(* Logix 5000 project; controller R5_CSS vendor 1 type 14 code 74 rev 19.11; software revision 19.01; part 5 of 18 *)
(* tags used below, declared in another part *)
   Coal_Tank_Heel_Inches : REAL;
   Coal_Tank_Height_Inches : REAL;
   ColdBoot : BOOL;
   DisableCommand : BOOL;
   EnableCommand : BOOL;
   Fault : BOOL;
   FirstScanLatch : BOOL;
   FirstScanLatchTON : TIMER;
   HART1 : HARTModuleDef;
   HARTData1 : HARTData;
   HEART_DATA : INT[122];
   IP_Address : DINT[4];
   IP_AddressGetMSG : MESSAGE;
   IP_AddressGetMSG_TON : TIMER;
   IP_AddressSetMSG : MESSAGE;
   LC303A : LEVEL_CONTROL;   // AQUEOUS PHASE OF PRIMARY SETTLER
   LC303A_LT_Raw : REAL;
   LC303B : LEVEL_CONTROL;   // INTERFACE LEVEL OF PRIMARY CONDENSER
   LC303B_LT_Raw : REAL;
   LT303_Probe_Length_Inches : REAL;
   LT303_RAW : REAL[5];   // LT 303 RAW
   LT303_Scale_Param : REAL;
   My_IP_Address : DINT[4];
   My_Subnet : DINT[4];
   P101A : PUMP_CONTROL;
   P101B : PUMP_CONTROL;
   P303A : PUMP_CONTROL;
   P303B : PUMP_CONTROL;
   SetMyIP_Enabled : BOOL;
   TCP_GetAll : TCPGetAllConfig;
   TCP_SetAll : TCPSetAllConfig;
   Test : INT[500];
   WarmBoot : BOOL;
(* MainProgram, continued *)

ROUTINE A2a_MM_HART   (* ladder *)
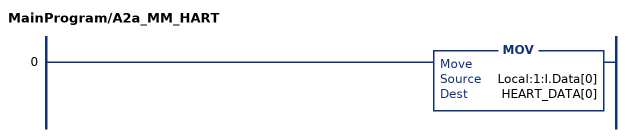
   0: MOV(Local:1:I.Data[0],HEART_DATA[0]);
END_ROUTINE

ROUTINE A2b_HART_READ   (* ladder *)
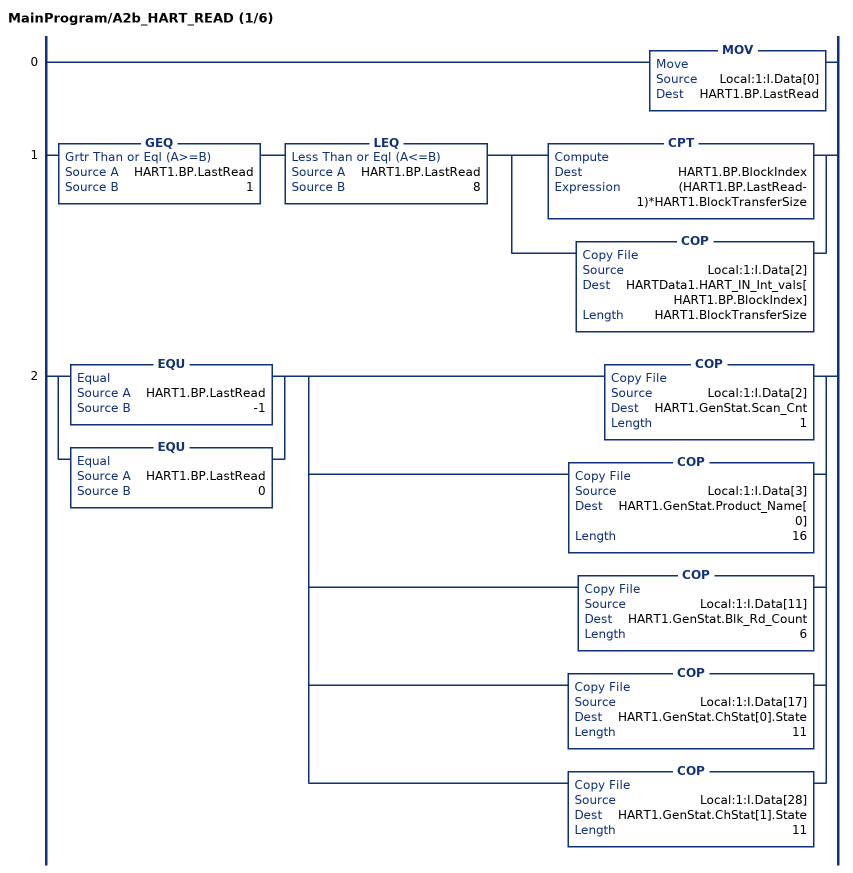
   0: MOV(Local:1:I.Data[0],HART1.BP.LastRead);
   1: GEQ(HART1.BP.LastRead,1)LEQ(HART1.BP.LastRead,8)[CPT(HART1.BP.BlockIndex,(HART1.BP.LastRead-1)*HART1.BlockTransferSize) ,COP(Local:1:I.Data[2],HARTData1.HART_IN_Int_vals[HART1.BP.BlockIndex],HART1.BlockTransferSize) ];
   2: [EQU(HART1.BP.LastRead,-1) ,EQU(HART1.BP.LastRead,0) ][COP(Local:1:I.Data[2],HART1.GenStat.Scan_Cnt,1) ,COP(Local:1:I.Data[3],HART1.GenStat.Product_Name[0],16) ,COP(Local:1:I.Data[11],HART1.GenStat.Blk_Rd_Count,6) ,COP(Local:1:I.Data[17],HART1.GenStat.ChStat[0].State,11) ,COP(Local:1:I.Data[28],HART1.GenStat.ChStat[1].State,11) ];
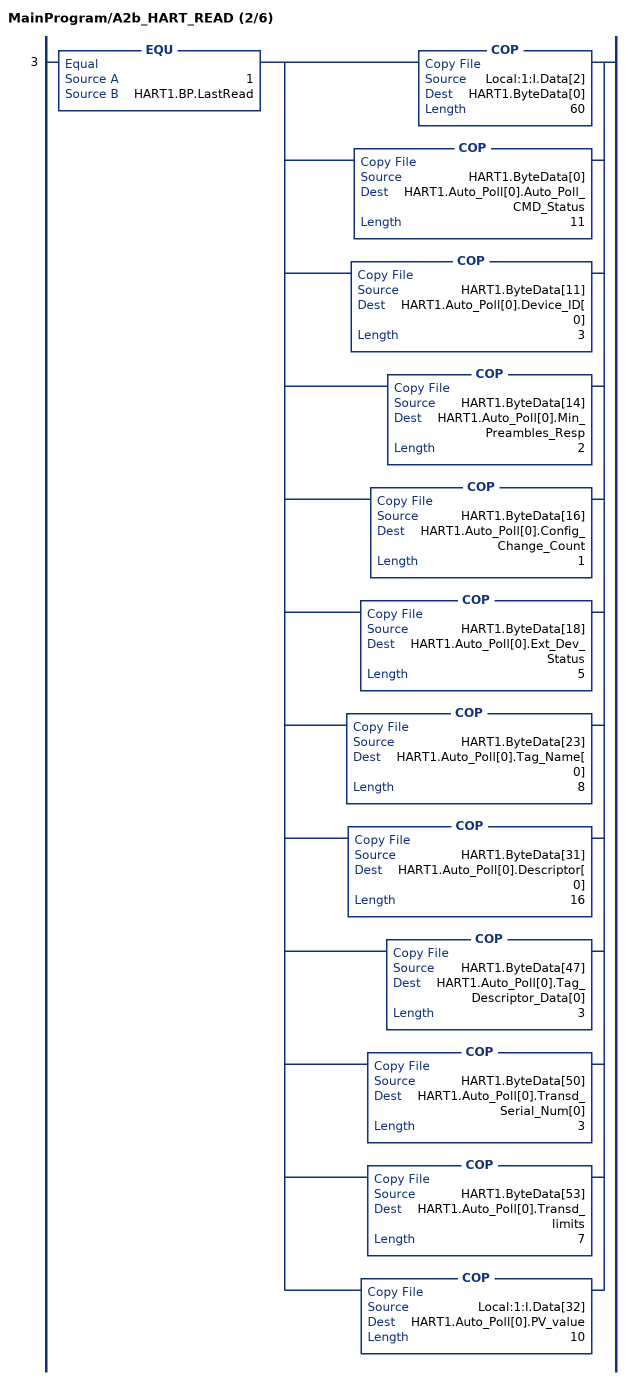
   3: EQU(1,HART1.BP.LastRead)[COP(Local:1:I.Data[2],HART1.ByteData[0],60) ,COP(HART1.ByteData[0],HART1.Auto_Poll[0].Auto_Poll_CMD_Status,11) ,COP(HART1.ByteData[11],HART1.Auto_Poll[0].Device_ID[0],3) ,COP(HART1.ByteData[14],HART1.Auto_Poll[0].Min_Preambles_Resp,2) ,COP(HART1.ByteData[16],HART1.Auto_Poll[0].Config_Change_Count,1) ,COP(HART1.ByteData[18],HART1.Auto_Poll[0].Ext_Dev_Status,5) ,COP(HART1.ByteData[23],HART1.Auto_Poll[0].Tag_Name[0],8) ,COP(HART1.ByteData[31],HART1.Auto_Poll[0].Descriptor[0],16) ,COP(HART1.ByteData[47],HART1.Auto_Poll[0].Tag_Descriptor_Data[0],3) ,COP(HART1.ByteData[50],HART1.Auto_Poll[0].Transd_Serial_Num[0],3) ,COP(HART1.ByteData[53],HART1.Auto_Poll[0].Transd_limits,7) ,COP(Local:1:I.Data[32],HART1.Auto_Poll[0].PV_value,10) ];
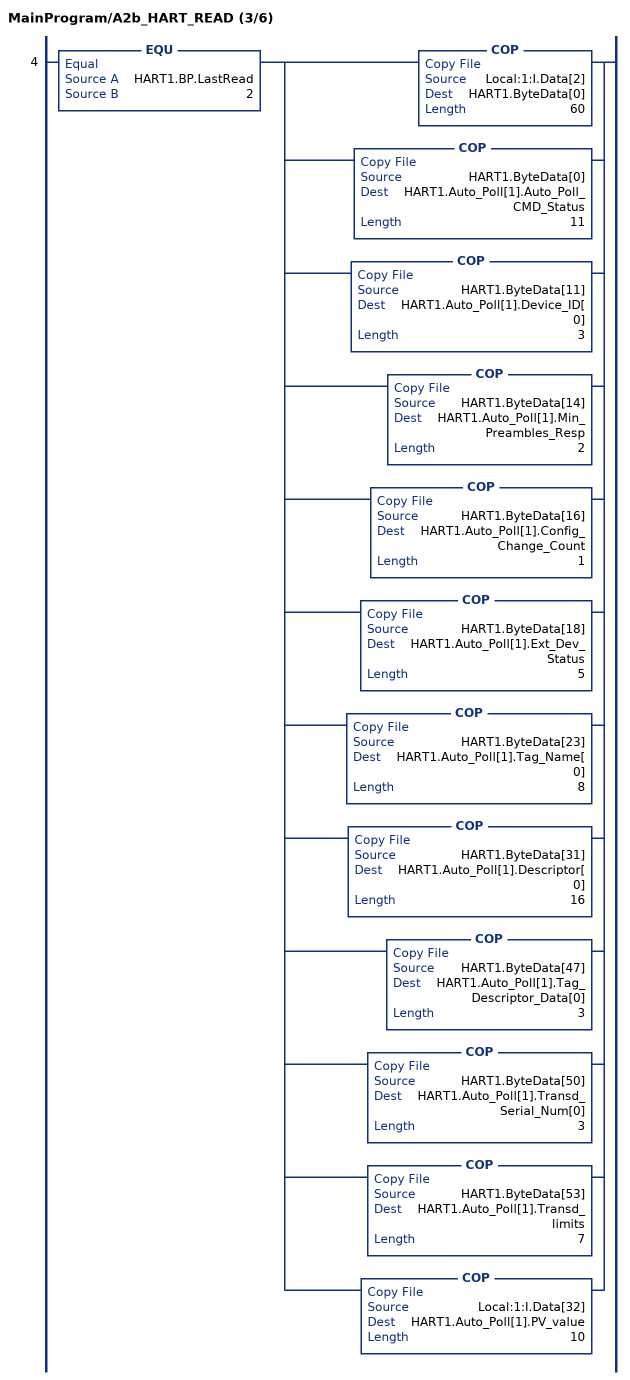
   4: EQU(HART1.BP.LastRead,2)[COP(Local:1:I.Data[2],HART1.ByteData[0],60) ,COP(HART1.ByteData[0],HART1.Auto_Poll[1].Auto_Poll_CMD_Status,11) ,COP(HART1.ByteData[11],HART1.Auto_Poll[1].Device_ID[0],3) ,COP(HART1.ByteData[14],HART1.Auto_Poll[1].Min_Preambles_Resp,2) ,COP(HART1.ByteData[16],HART1.Auto_Poll[1].Config_Change_Count,1) ,COP(HART1.ByteData[18],HART1.Auto_Poll[1].Ext_Dev_Status,5) ,COP(HART1.ByteData[23],HART1.Auto_Poll[1].Tag_Name[0],8) ,COP(HART1.ByteData[31],HART1.Auto_Poll[1].Descriptor[0],16) ,COP(HART1.ByteData[47],HART1.Auto_Poll[1].Tag_Descriptor_Data[0],3) ,COP(HART1.ByteData[50],HART1.Auto_Poll[1].Transd_Serial_Num[0],3) ,COP(HART1.ByteData[53],HART1.Auto_Poll[1].Transd_limits,7) ,COP(Local:1:I.Data[32],HART1.Auto_Poll[1].PV_value,10) ];
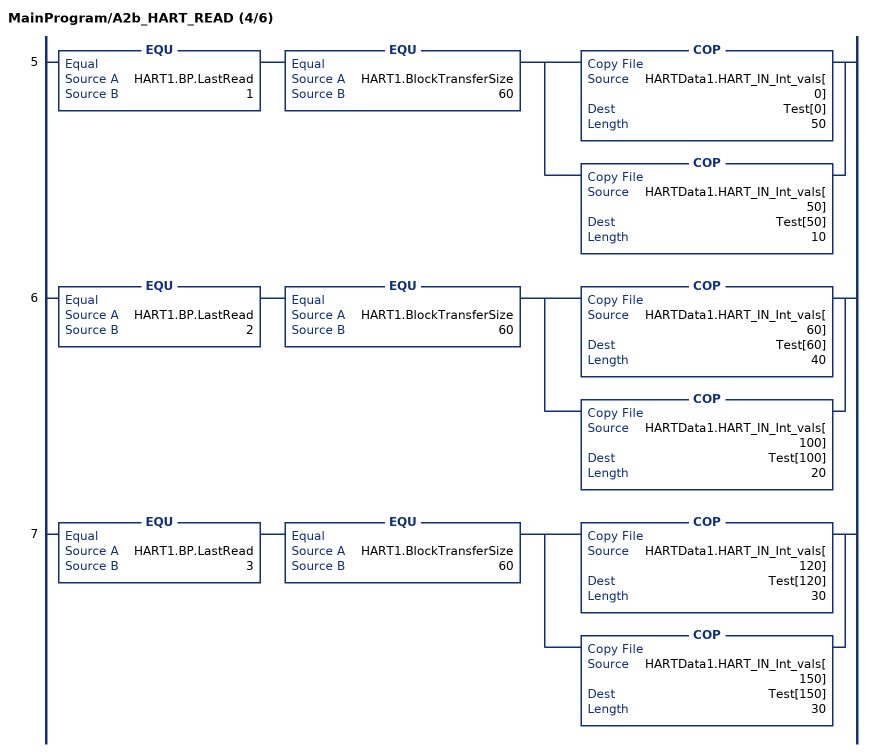
   5: EQU(HART1.BP.LastRead,1)EQU(HART1.BlockTransferSize,60)[COP(HARTData1.HART_IN_Int_vals[0],Test[0],50) ,COP(HARTData1.HART_IN_Int_vals[50],Test[50],10) ];
   6: EQU(HART1.BP.LastRead,2)EQU(HART1.BlockTransferSize,60)[COP(HARTData1.HART_IN_Int_vals[60],Test[60],40) ,COP(HARTData1.HART_IN_Int_vals[100],Test[100],20) ];
   7: EQU(HART1.BP.LastRead,3)EQU(HART1.BlockTransferSize,60)[COP(HARTData1.HART_IN_Int_vals[120],Test[120],30) ,COP(HARTData1.HART_IN_Int_vals[150],Test[150],30) ];
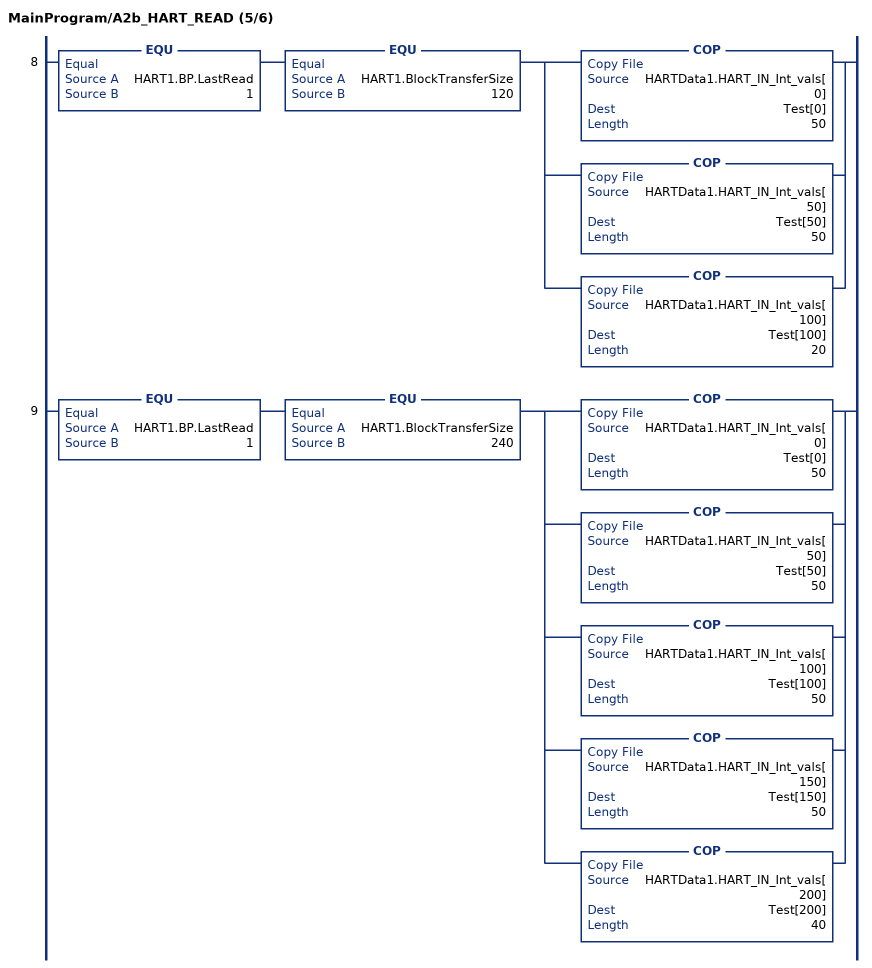
   8: EQU(HART1.BP.LastRead,1)EQU(HART1.BlockTransferSize,120)[COP(HARTData1.HART_IN_Int_vals[0],Test[0],50) ,COP(HARTData1.HART_IN_Int_vals[50],Test[50],50) ,COP(HARTData1.HART_IN_Int_vals[100],Test[100],20) ];
   9: EQU(HART1.BP.LastRead,1)EQU(HART1.BlockTransferSize,240)[COP(HARTData1.HART_IN_Int_vals[0],Test[0],50) ,COP(HARTData1.HART_IN_Int_vals[50],Test[50],50) ,COP(HARTData1.HART_IN_Int_vals[100],Test[100],50) ,COP(HARTData1.HART_IN_Int_vals[150],Test[150],50) ,COP(HARTData1.HART_IN_Int_vals[200],Test[200],40) ];
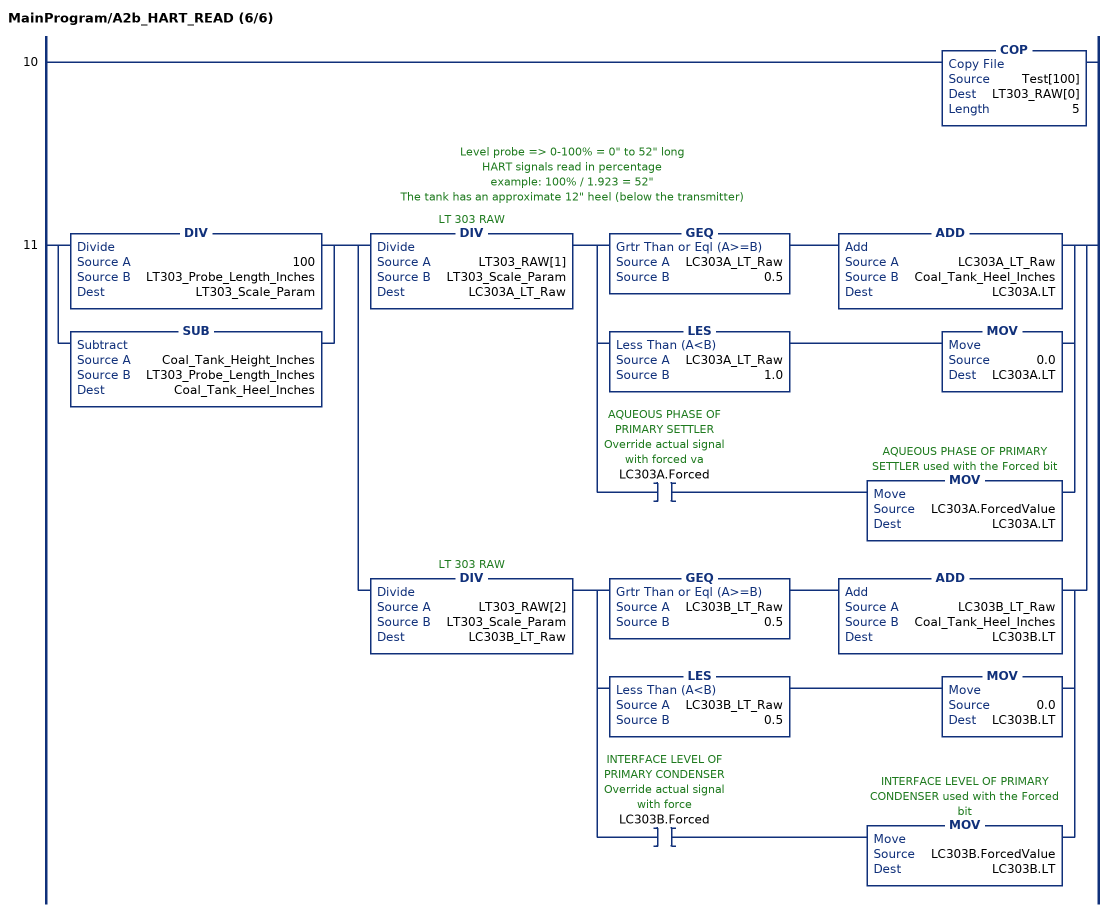
   10: COP(Test[100],LT303_RAW[0],5);
   // Level probe => 0-100% = 0" to 52" long
   // HART signals read in percentage
   // example: 100% / 1.923 = 52"
   // The tank has an approximate 12" heel (below the transmitter)
   11: [DIV(100,LT303_Probe_Length_Inches,LT303_Scale_Param) ,SUB(Coal_Tank_Height_Inches,LT303_Probe_Length_Inches,Coal_Tank_Heel_Inches) ][DIV(LT303_RAW[1],LT303_Scale_Param,LC303A_LT_Raw) [GEQ(LC303A_LT_Raw,0.5) ADD(LC303A_LT_Raw,Coal_Tank_Heel_Inches,LC303A.LT) ,LES(LC303A_LT_Raw,1.0) MOV(0.0,LC303A.LT) ,XIC(LC303A.Forced) MOV(LC303A.ForcedValue,LC303A.LT) ] ,DIV(LT303_RAW[2],LT303_Scale_Param,LC303B_LT_Raw) [GEQ(LC303B_LT_Raw,0.5) ADD(LC303B_LT_Raw,Coal_Tank_Heel_Inches,LC303B.LT) ,LES(LC303B_LT_Raw,0.5) MOV(0.0,LC303B.LT) ,XIC(LC303B.Forced) MOV(LC303B.ForcedValue,LC303B.LT) ] ];
END_ROUTINE

ROUTINE A2c_HART_WRITEE   (* ladder *)
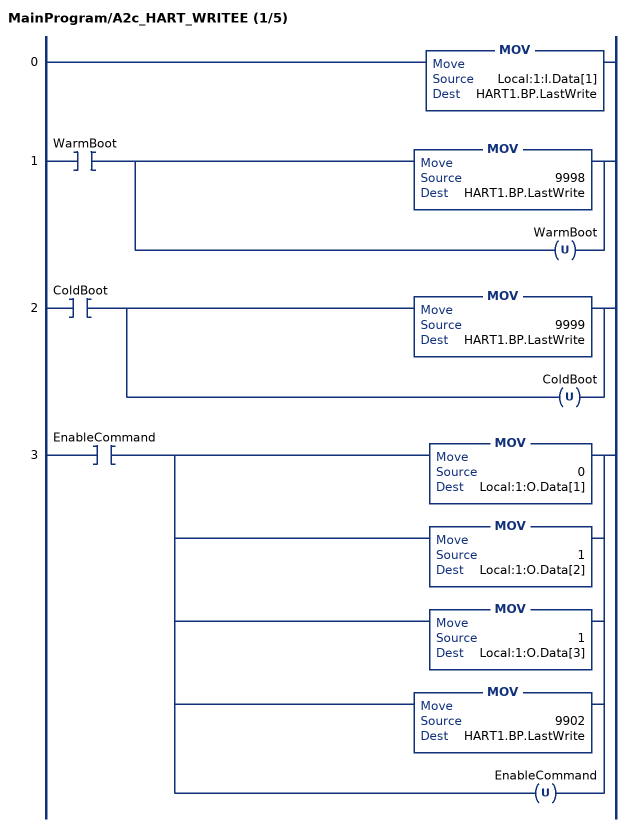
   0: MOV(Local:1:I.Data[1],HART1.BP.LastWrite);
   1: XIC(WarmBoot)[MOV(9998,HART1.BP.LastWrite) ,OTU(WarmBoot) ];
   2: XIC(ColdBoot)[MOV(9999,HART1.BP.LastWrite) ,OTU(ColdBoot) ];
   3: XIC(EnableCommand)[MOV(0,Local:1:O.Data[1]) ,MOV(1,Local:1:O.Data[2]) ,MOV(1,Local:1:O.Data[3]) ,MOV(9902,HART1.BP.LastWrite) ,OTU(EnableCommand) ];
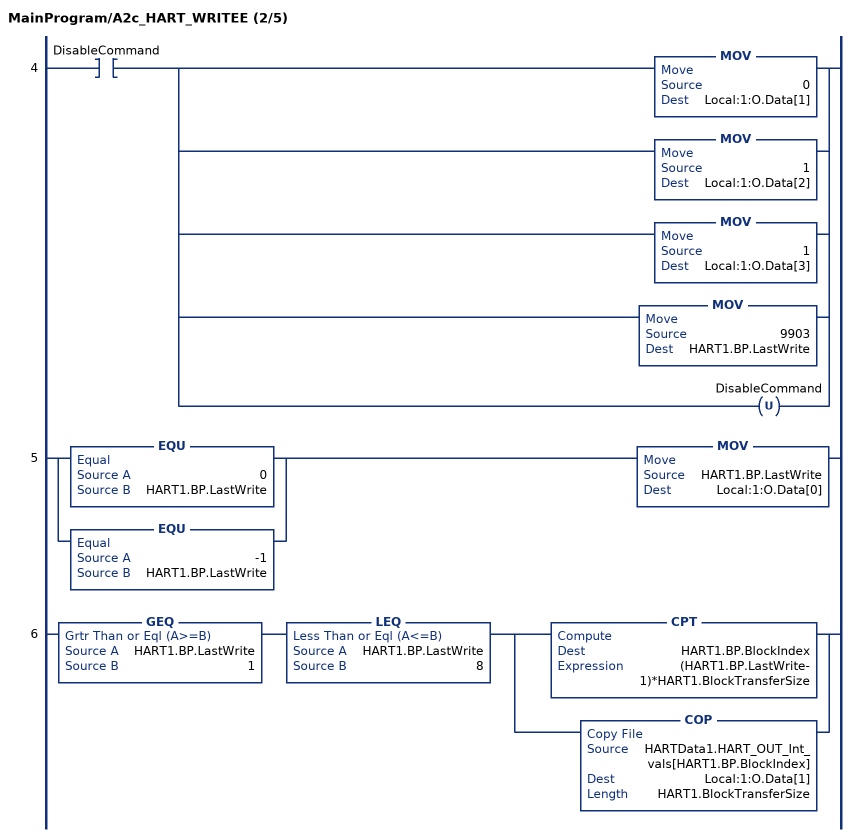
   4: XIC(DisableCommand)[MOV(0,Local:1:O.Data[1]) ,MOV(1,Local:1:O.Data[2]) ,MOV(1,Local:1:O.Data[3]) ,MOV(9903,HART1.BP.LastWrite) ,OTU(DisableCommand) ];
   5: [EQU(0,HART1.BP.LastWrite) ,EQU(-1,HART1.BP.LastWrite) ]MOV(HART1.BP.LastWrite,Local:1:O.Data[0]);
   6: GEQ(HART1.BP.LastWrite,1)LEQ(HART1.BP.LastWrite,8)[CPT(HART1.BP.BlockIndex,(HART1.BP.LastWrite-1)*HART1.BlockTransferSize) ,COP(HARTData1.HART_OUT_Int_vals[HART1.BP.BlockIndex],Local:1:O.Data[1],HART1.BlockTransferSize) ];
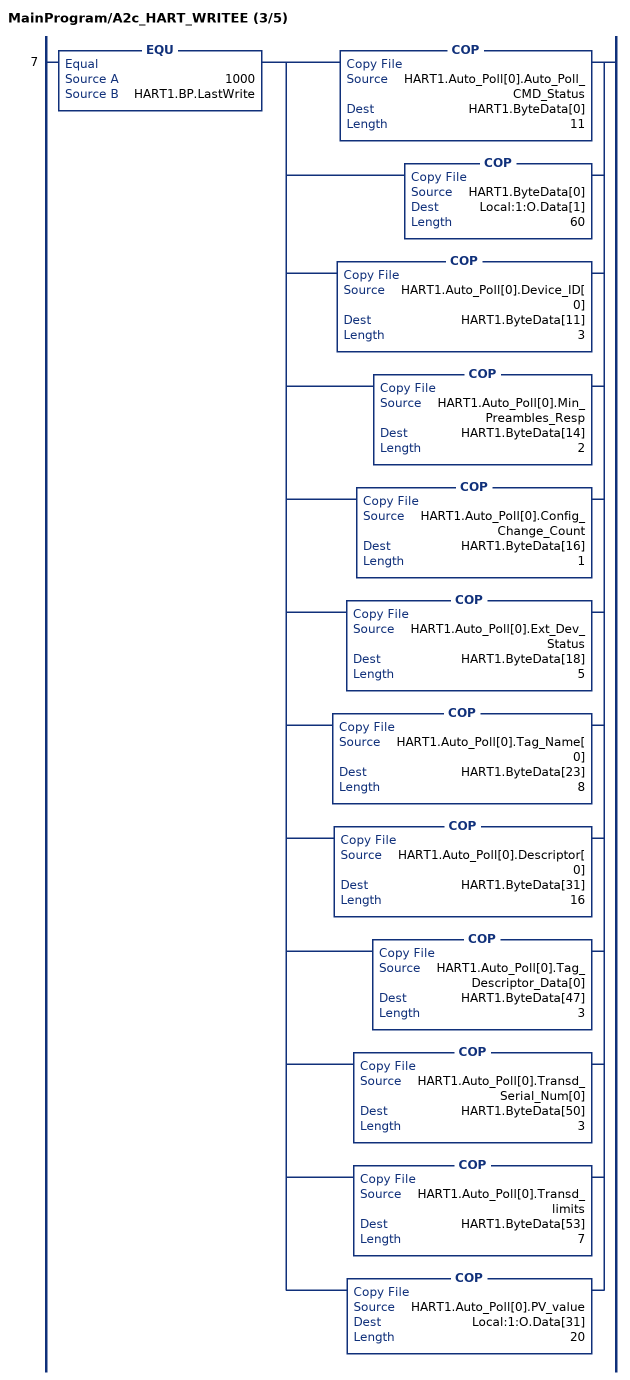
   7: EQU(1000,HART1.BP.LastWrite)[COP(HART1.Auto_Poll[0].Auto_Poll_CMD_Status,HART1.ByteData[0],11) ,COP(HART1.ByteData[0],Local:1:O.Data[1],60) ,COP(HART1.Auto_Poll[0].Device_ID[0],HART1.ByteData[11],3) ,COP(HART1.Auto_Poll[0].Min_Preambles_Resp,HART1.ByteData[14],2) ,COP(HART1.Auto_Poll[0].Config_Change_Count,HART1.ByteData[16],1) ,COP(HART1.Auto_Poll[0].Ext_Dev_Status,HART1.ByteData[18],5) ,COP(HART1.Auto_Poll[0].Tag_Name[0],HART1.ByteData[23],8) ,COP(HART1.Auto_Poll[0].Descriptor[0],HART1.ByteData[31],16) ,COP(HART1.Auto_Poll[0].Tag_Descriptor_Data[0],HART1.ByteData[47],3) ,COP(HART1.Auto_Poll[0].Transd_Serial_Num[0],HART1.ByteData[50],3) ,COP(HART1.Auto_Poll[0].Transd_limits,HART1.ByteData[53],7) ,COP(HART1.Auto_Poll[0].PV_value,Local:1:O.Data[31],20) ];
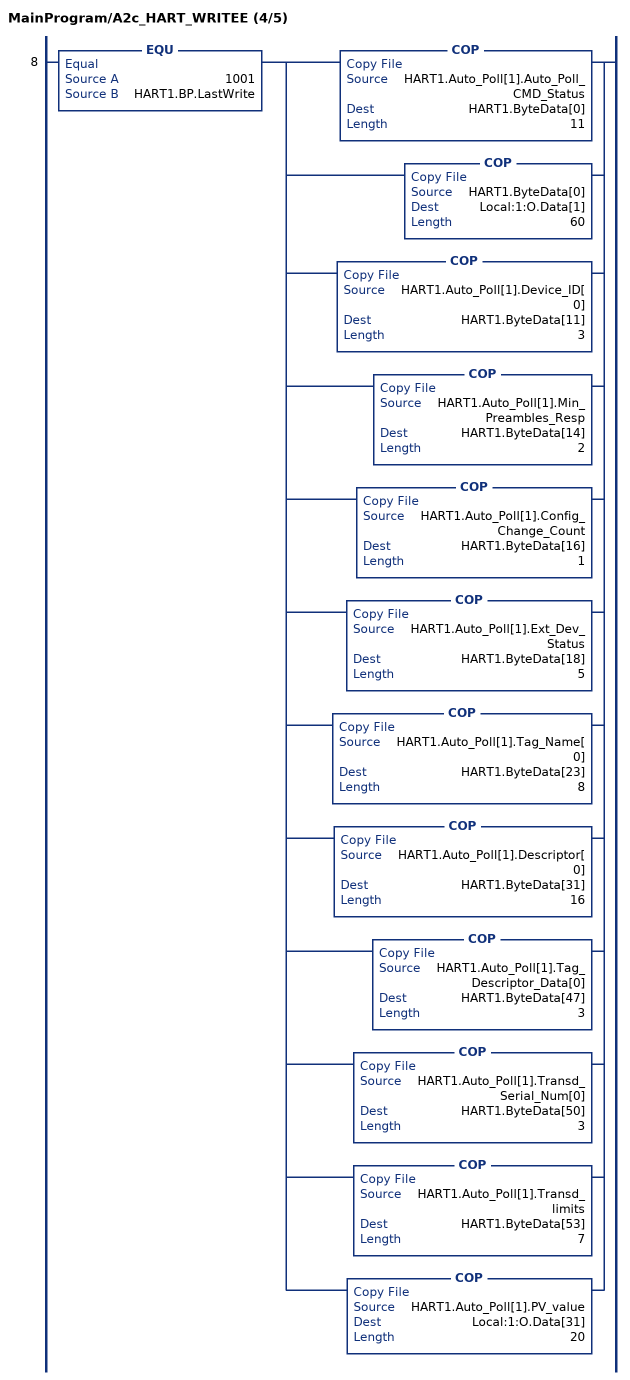
   8: EQU(1001,HART1.BP.LastWrite)[COP(HART1.Auto_Poll[1].Auto_Poll_CMD_Status,HART1.ByteData[0],11) ,COP(HART1.ByteData[0],Local:1:O.Data[1],60) ,COP(HART1.Auto_Poll[1].Device_ID[0],HART1.ByteData[11],3) ,COP(HART1.Auto_Poll[1].Min_Preambles_Resp,HART1.ByteData[14],2) ,COP(HART1.Auto_Poll[1].Config_Change_Count,HART1.ByteData[16],1) ,COP(HART1.Auto_Poll[1].Ext_Dev_Status,HART1.ByteData[18],5) ,COP(HART1.Auto_Poll[1].Tag_Name[0],HART1.ByteData[23],8) ,COP(HART1.Auto_Poll[1].Descriptor[0],HART1.ByteData[31],16) ,COP(HART1.Auto_Poll[1].Tag_Descriptor_Data[0],HART1.ByteData[47],3) ,COP(HART1.Auto_Poll[1].Transd_Serial_Num[0],HART1.ByteData[50],3) ,COP(HART1.Auto_Poll[1].Transd_limits,HART1.ByteData[53],7) ,COP(HART1.Auto_Poll[1].PV_value,Local:1:O.Data[31],20) ];
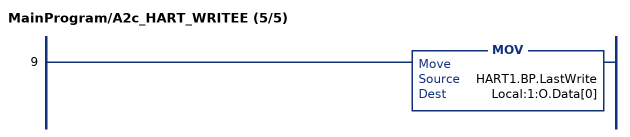
   9: MOV(HART1.BP.LastWrite,Local:1:O.Data[0]);
END_ROUTINE

ROUTINE A3_ENET_STATUS   (* ladder *)
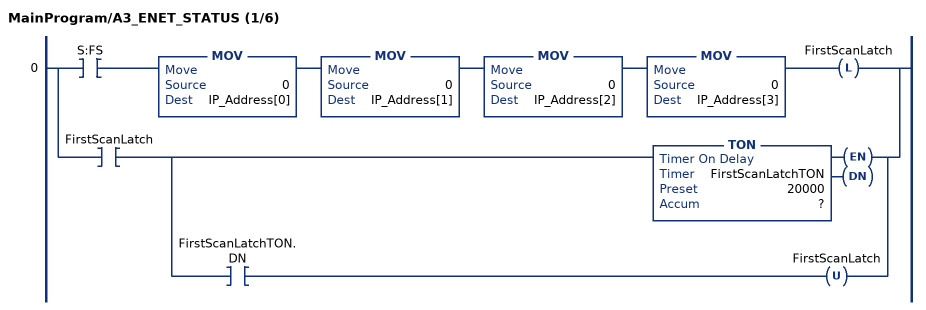
   0: [XIC(S:FS) MOV(0,IP_Address[0]) MOV(0,IP_Address[1]) MOV(0,IP_Address[2]) MOV(0,IP_Address[3]) OTL(FirstScanLatch) ,XIC(FirstScanLatch) [TON(FirstScanLatchTON,?,?) ,XIC(FirstScanLatchTON.DN) OTU(FirstScanLatch) ] ];
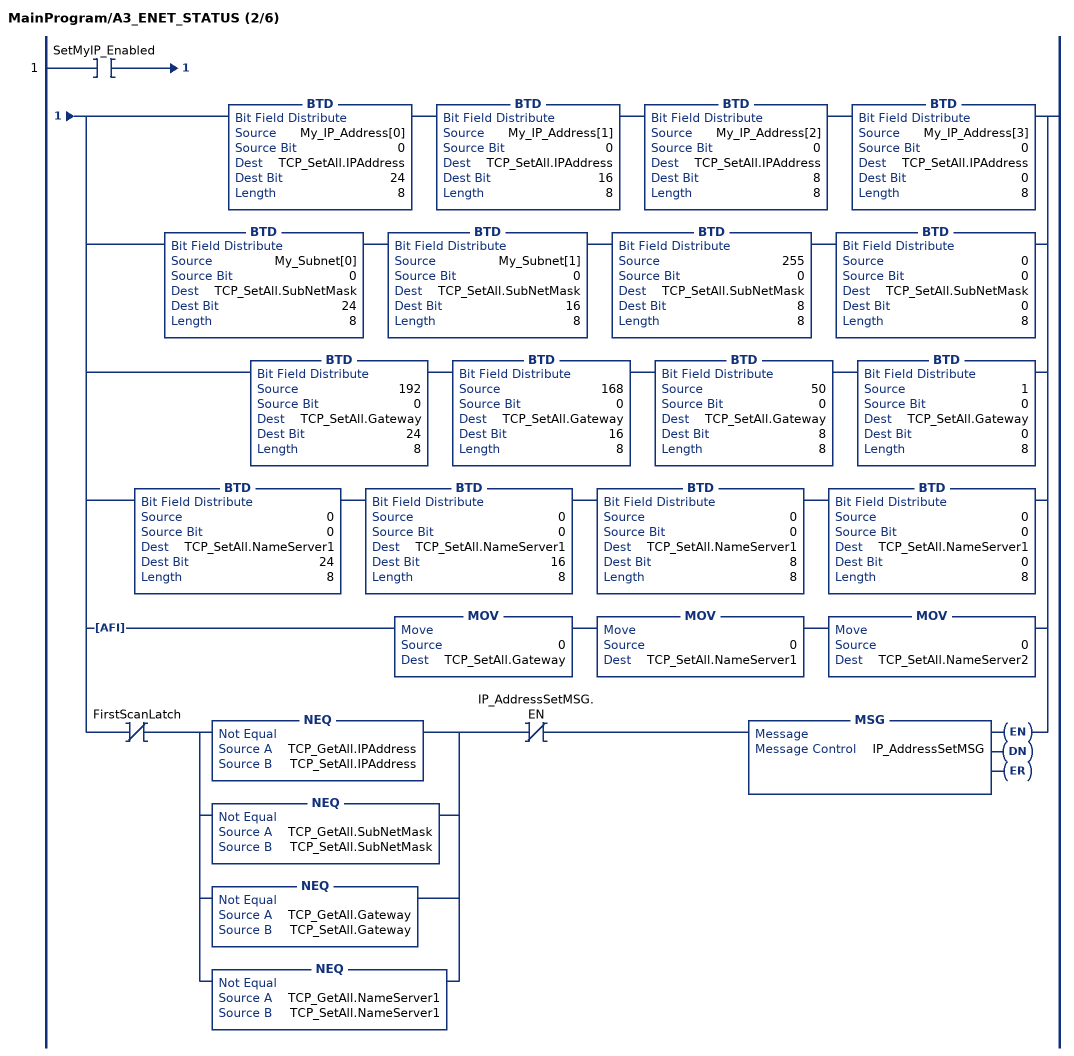
   1: XIC(SetMyIP_Enabled)[BTD(My_IP_Address[0],0,TCP_SetAll.IPAddress,24,8) BTD(My_IP_Address[1],0,TCP_SetAll.IPAddress,16,8) BTD(My_IP_Address[2],0,TCP_SetAll.IPAddress,8,8) BTD(My_IP_Address[3],0,TCP_SetAll.IPAddress,0,8) ,BTD(My_Subnet[0],0,TCP_SetAll.SubNetMask,24,8) BTD(My_Subnet[1],0,TCP_SetAll.SubNetMask,16,8) BTD(255,0,TCP_SetAll.SubNetMask,8,8) BTD(0,0,TCP_SetAll.SubNetMask,0,8) ,BTD(192,0,TCP_SetAll.Gateway,24,8) BTD(168,0,TCP_SetAll.Gateway,16,8) BTD(50,0,TCP_SetAll.Gateway,8,8) BTD(1,0,TCP_SetAll.Gateway,0,8) ,BTD(0,0,TCP_SetAll.NameServer1,24,8) BTD(0,0,TCP_SetAll.NameServer1,16,8) BTD(0,0,TCP_SetAll.NameServer1,8,8) BTD(0,0,TCP_SetAll.NameServer1,0,8) ,AFI() MOV(0,TCP_SetAll.Gateway) MOV(0,TCP_SetAll.NameServer1) MOV(0,TCP_SetAll.NameServer2) ,XIO(FirstScanLatch) [NEQ(TCP_GetAll.IPAddress,TCP_SetAll.IPAddress) ,NEQ(TCP_GetAll.SubNetMask,TCP_SetAll.SubNetMask) ,NEQ(TCP_GetAll.Gateway,TCP_SetAll.Gateway) ,NEQ(TCP_GetAll.NameServer1,TCP_SetAll.NameServer1) ] XIO(IP_AddressSetMSG.EN) MSG(IP_AddressSetMSG) ];
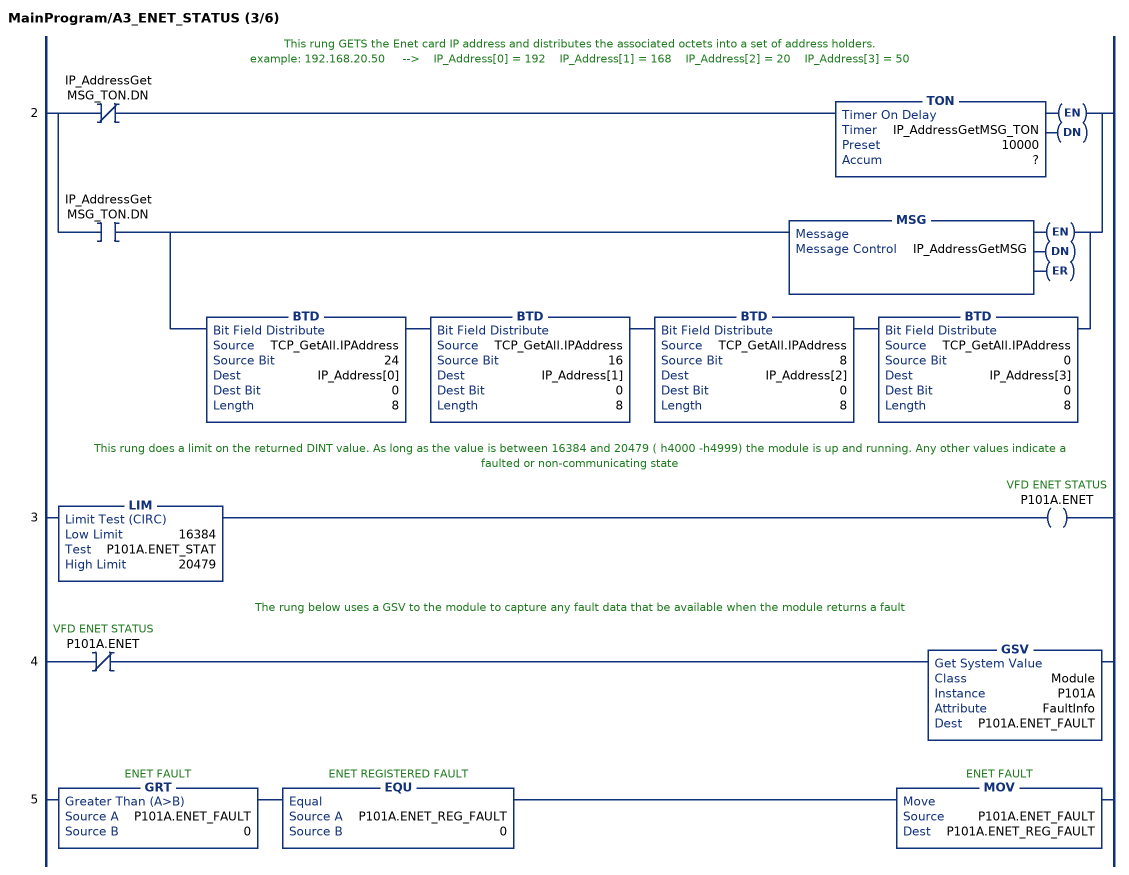
   // This rung GETS the Enet card IP address and distributes the associated octets into a set of address holders.
   // example: 192.168.20.50     -->    IP_Address[0] = 192    IP_Address[1] = 168    IP_Address[2] = 20    IP_Address[3] = 50
   2: [XIO(IP_AddressGetMSG_TON.DN) TON(IP_AddressGetMSG_TON,?,?) ,XIC(IP_AddressGetMSG_TON.DN) [MSG(IP_AddressGetMSG) ,BTD(TCP_GetAll.IPAddress,24,IP_Address[0],0,8) BTD(TCP_GetAll.IPAddress,16,IP_Address[1],0,8) BTD(TCP_GetAll.IPAddress,8,IP_Address[2],0,8) BTD(TCP_GetAll.IPAddress,0,IP_Address[3],0,8) ] ];
   // This rung does a limit on the returned DINT value. As long as the value is between 16384 and 20479 ( h4000 -h4999) the module is up and running. Any other values indicate a faulted or non-communicating state
   3: LIM(16384,P101A.ENET_STAT,20479)OTE(P101A.ENET);
   // The rung below uses a GSV to the module to capture any fault data that be available when the module returns a fault
   4: XIO(P101A.ENET)GSV(Module,P101A,FaultInfo,P101A.ENET_FAULT);
   5: GRT(P101A.ENET_FAULT,0)EQU(P101A.ENET_REG_FAULT,0)MOV(P101A.ENET_FAULT,P101A.ENET_REG_FAULT);
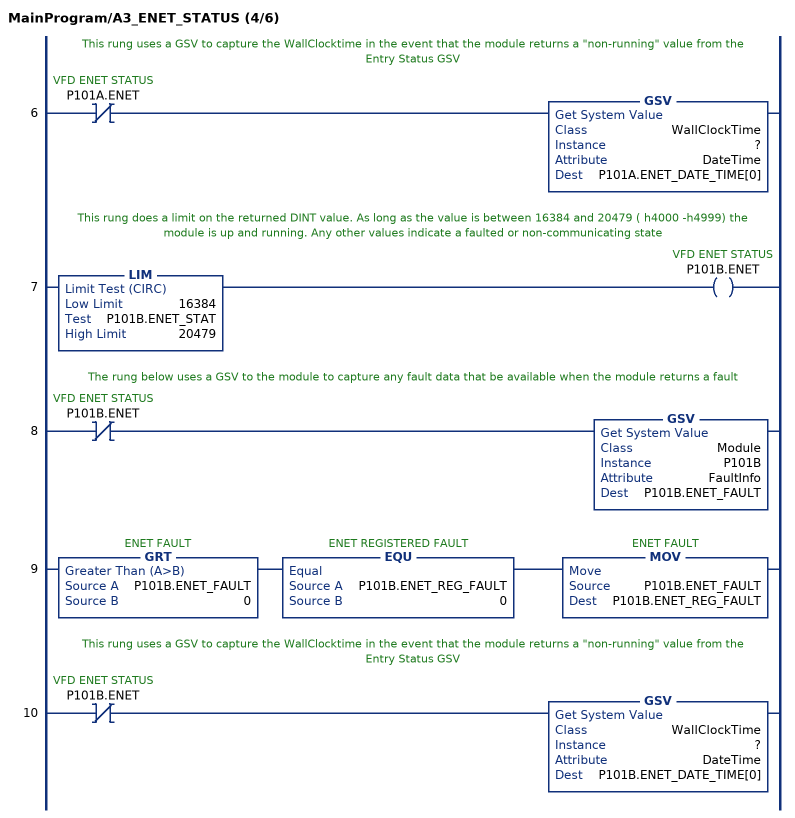
   // This rung uses a GSV to capture the WallClocktime in the event that the module returns a "non-running" value from the Entry Status GSV
   6: XIO(P101A.ENET)GSV(WallClockTime,?,DateTime,P101A.ENET_DATE_TIME[0]);
   // This rung does a limit on the returned DINT value. As long as the value is between 16384 and 20479 ( h4000 -h4999) the module is up and running. Any other values indicate a faulted or non-communicating state
   7: LIM(16384,P101B.ENET_STAT,20479)OTE(P101B.ENET);
   // The rung below uses a GSV to the module to capture any fault data that be available when the module returns a fault
   8: XIO(P101B.ENET)GSV(Module,P101B,FaultInfo,P101B.ENET_FAULT);
   9: GRT(P101B.ENET_FAULT,0)EQU(P101B.ENET_REG_FAULT,0)MOV(P101B.ENET_FAULT,P101B.ENET_REG_FAULT);
   // This rung uses a GSV to capture the WallClocktime in the event that the module returns a "non-running" value from the Entry Status GSV
   10: XIO(P101B.ENET)GSV(WallClockTime,?,DateTime,P101B.ENET_DATE_TIME[0]);
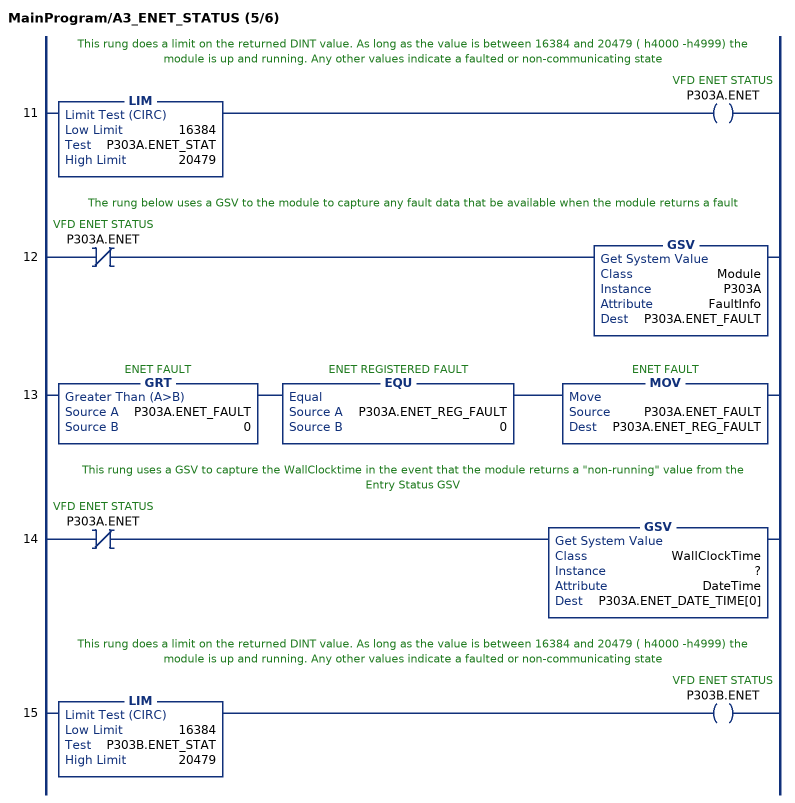
   // This rung does a limit on the returned DINT value. As long as the value is between 16384 and 20479 ( h4000 -h4999) the module is up and running. Any other values indicate a faulted or non-communicating state
   11: LIM(16384,P303A.ENET_STAT,20479)OTE(P303A.ENET);
   // The rung below uses a GSV to the module to capture any fault data that be available when the module returns a fault
   12: XIO(P303A.ENET)GSV(Module,P303A,FaultInfo,P303A.ENET_FAULT);
   13: GRT(P303A.ENET_FAULT,0)EQU(P303A.ENET_REG_FAULT,0)MOV(P303A.ENET_FAULT,P303A.ENET_REG_FAULT);
   // This rung uses a GSV to capture the WallClocktime in the event that the module returns a "non-running" value from the Entry Status GSV
   14: XIO(P303A.ENET)GSV(WallClockTime,?,DateTime,P303A.ENET_DATE_TIME[0]);
   // This rung does a limit on the returned DINT value. As long as the value is between 16384 and 20479 ( h4000 -h4999) the module is up and running. Any other values indicate a faulted or non-communicating state
   15: LIM(16384,P303B.ENET_STAT,20479)OTE(P303B.ENET);
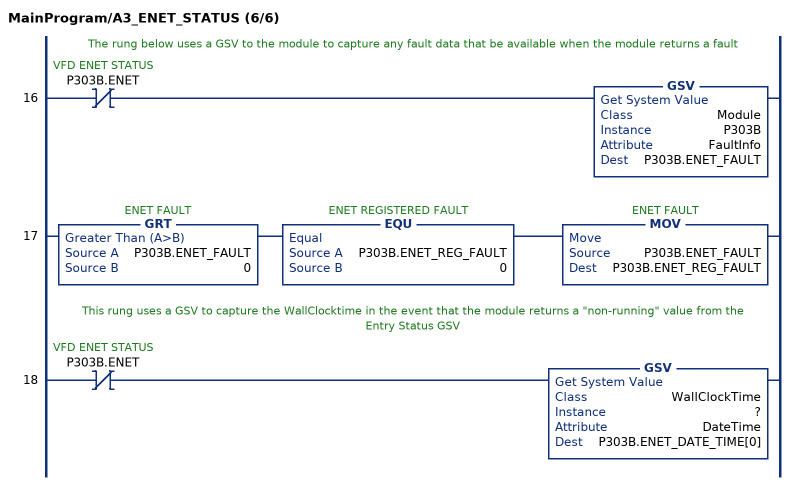
   // The rung below uses a GSV to the module to capture any fault data that be available when the module returns a fault
   16: XIO(P303B.ENET)GSV(Module,P303B,FaultInfo,P303B.ENET_FAULT);
   17: GRT(P303B.ENET_FAULT,0)EQU(P303B.ENET_REG_FAULT,0)MOV(P303B.ENET_FAULT,P303B.ENET_REG_FAULT);
   // This rung uses a GSV to capture the WallClocktime in the event that the module returns a "non-running" value from the Entry Status GSV
   18: XIO(P303B.ENET)GSV(WallClockTime,?,DateTime,P303B.ENET_DATE_TIME[0]);
END_ROUTINE
